//This function is used to calculate the gap size between two 'barn door' type blades
FUNCTION_BLOCK FB_CalculateGap

VAR_INPUT

AngleBladeA : LREAL;
AngleBladeB : LREAL;
fBladeSize : LREAL:=62.94;
fClosedGap : LREAL:=2.00;
ENC_CONSTANT : LREAL;
END_VAR

VAR_OUTPUT

GapSize : LREAL;
iGapSize AT %Q* : DINT;

END_VAR

VAR



END_VAR

GapSize := fClosedGap + fBladeSize*(2-(COS(DEG_TO_RAD(AngleBladeA)) + COS(DEG_TO_RAD(AngleBladeB))));
iGapSize := REAL_TO_DINT(GapSize * ENC_CONSTANT);

END_FUNCTION_BLOCK

(* stored: Version 1.1.0.1, ProductVersion 3.1.4024.0
   POU FB_CalculateGap: Id {eb587f1b-0364-468c-9da3-6eac971ef0df}, SpecialFunc None *)
